PROGRAM MAIN
VAR
		// stepper function blocks  
	mcPower_1 : MC_Power;
	mcReset_1 : MC_Reset;
	mcJogging_1 : MC_Jog;
	mcMoveAbs_1 : MC_MoveAbsolute;
	mcMoveRel_1 : MC_MoveRelative;
	mcStop : MC_Stop;
	mcHome_1 : MC_Home;
	
	bEnableAxis_1 : BOOL;
	bJogForwards : BOOL;
	bJogBackwards: BOOL;
	eJogMode : E_JogMode; 
	bMoveDone : BOOL;	
	bAbsMove: BOOL;
	bRelMove: BOOL;
	
	heartbeat: BYTE; 
	//FbStageMotion : FB_Stage_Motion;

	bStop: BOOL;
	bHomeAxis_1: BOOL;

	// action Variables
	mcMoveAbsTest_1 : MC_MoveAbsolute;
	mcMoveAbsTestReturn_1 : MC_MoveAbsolute;
	iState : DINT;
	bStartTest : BOOL;
	bFinishTest: BOOL;
	fbReturnTimer : TON; // timer delay for the cycle to return home.
	fbDutyCycleTimer : TON; // timer duty cycle so the delay between cycles
	bStartReturnTimer : BOOL;
	bStartDutyCycleTimer : BOOL;	
	fbTestCycleCounter  : CTU;
	bCycleComplete : BOOL;
	bCycleCounterReset : BOOL;
	bTestFinished : BOOL;
	bTestRelMove: BOOL;
	
	bEnableAxisPosative_1: BOOL;
	bEnableAxisNegative_1: BOOL;
END_VAR

VAR_INPUT
	fAbsPos_1: LREAL;
	fRelDistance: LREAL;
	fRelTestDistance: LREAL;
	fAbsTestDistance: LREAL;
	fHomePosition: LREAL;
	fAxisVelocity: LREAL;
	fAxisAcceleration: LREAL;
	
// action Variables
	iCycleCount : WORD;
	fReturnTime : TIME;
	uInputReurnTime : UINT;
	fDutyCycleTime : TIME;
	uInputCycleTime : UINT;
	fTempLimit : DINT;
	
// Digital Inputs
	LimitSwitchInput_1 AT %I* : BOOL;
	LimitSwitchInput_2 AT %I* : BOOL;
	
// Analouge Inputs
	ThermoCoupleValue_Ch1 AT %I* : DINT;  
END_VAR

VAR_OUTPUT
// action Variables	
	iCurrentCycleValue : WORD;
		// Digital outputs
	LimitSwitchOutput_1 AT %Q* : BOOL;
	LimitSwitchOutput_2 AT %Q* : BOOL;
	EncoderPowerOutput_3 AT %Q* : BOOL;
	EncoderPowerOutput_6 AT %Q* : BOOL;
END_VAR

heartbeat := heartbeat + 1;

Limit_Switch();
Thermo_Couple();
EncoderPowerOutput_3 := TRUE;
EncoderPowerOutput_6 := TRUE;

mcStop(Axis := GVL.stAxis_1, Execute := bStop,);

mcPower_1(Axis := GVL.stAxis_1, Enable := bEnableAxis_1, Enable_Positive := bEnableAxisPosative_1, Enable_Negative := bEnableAxisNegative_1, Override := 100.0);

mcReset_1(Axis := GVL.stAxis_1, Execute := NOT(bEnableAxis_1));

mcJogging_1(Axis := GVL.stAxis_1, JogForward := bJogForwards, JogBackwards := bJogBackwards, Velocity := fAxisVelocity, Acceleration := fAxisAcceleration, Deceleration := fAxisAcceleration, Jerk := 0.8);

mcMoveAbs_1 (Axis := GVL.stAxis_1, Execute := bAbsMove, Position := fAbsPos_1, Velocity := fAxisVelocity, Acceleration := fAxisAcceleration, Deceleration := fAxisAcceleration);
bAbsMove := FALSE;

mcMoveRel_1(Axis := GVL.stAxis_1, Execute := bRelMove, Distance := fRelDistance, Velocity := fAxisVelocity, Acceleration := fAxisAcceleration, Deceleration := fAxisAcceleration);
bRelMove := FALSE;

//mcHome_1(Axis := GVL.stAxis_1, Execute := bHomeAxis_1, Position := fHomePosition);


Test_Routine();

ACTION Limit_Switch:
LimitSwitchOutput_1 := TRUE;
LimitSwitchOutput_2 := TRUE;

IF LimitSwitchInput_1 THEN
	bEnableAxisPosative_1 := TRUE;
ELSE
	bEnableAxisPosative_1 := FALSE ;	
	
END_IF

IF LimitSwitchInput_2 THEN
	bEnableAxisNegative_1 := TRUE;
ELSE
	bEnableAxisNegative_1 := FALSE ;	
	
END_IF
END_ACTION

ACTION Test_Routine:
mcMoveAbsTest_1(Axis := GVL.stAxis_1, Position := 10, Velocity := fAxisVelocity, Acceleration := fAxisAcceleration, Deceleration := fAxisAcceleration);	
mcMoveAbsTest_1.Execute := FALSE;
fbReturnTimer( IN := bStartReturnTimer, PT := fReturnTime);	
mcMoveAbsTestReturn_1(Axis := GVL.stAxis_1, Position := 0, Velocity := fAxisVelocity, Acceleration := fAxisAcceleration, Deceleration := fAxisAcceleration);
mcMoveAbsTestReturn_1.Execute := FALSE;
fbReturnTimer( IN := bStartReturnTimer, PT := fReturnTime);	
fbDutyCycleTimer( IN := bStartDutyCycleTimer, PT := fDutyCycleTime);	
fbTestCycleCounter(CU := bCycleComplete, RESET := bCycleCounterReset, PV := iCycleCount);
fReturnTime:= INT_TO_TIME(uInputReurnTime);
fDutyCycleTime:= INT_TO_TIME(uInputCycleTime);
CASE iState OF
	
	// initialising the state machine so starting a homing rotuine reseting the counter to 0 
	0: 
		iState := 10;
	10: 
		IF bStartTest THEN
			iState := 20;
		END_IF
	
	20:
	
		mcMoveAbsTest_1.Execute := TRUE;
		IF mcMoveAbsTest_1.Done THEN
			bStartReturnTimer := TRUE;
			iState := 30;
		END_IF

	30:
		fbReturnTimer( IN := bStartReturnTimer, PT := fReturnTime);	
		IF MAIN.fbReturnTimer.Q THEN
			bStartReturnTimer := FALSE;
			iState := 40;
		END_IF
	

	40:
		mcMoveAbsTestReturn_1.Execute := TRUE;
		IF mcMoveAbsTestReturn_1.Done THEN
			bStartDutyCycleTimer := TRUE;
			iState := 50;
		END_IF	
	
	50:
		fbDutyCycleTimer( IN := bStartDutyCycleTimer, PT := fDutyCycleTime);	
		IF MAIN.fbDutyCycleTimer.Q THEN
			bStartDutyCycleTimer := FALSE;
			iState := 60;
		END_IF

	60: bCycleComplete := TRUE;
		iState := 70;
	
	70: fbTestCycleCounter(CU := bCycleComplete, RESET := bCycleCounterReset, PV := iCycleCount);
		IF MAIN.fbTestCycleCounter.Q THEN
			iState := 90; 
		ELSE
		bCycleComplete := FALSE;	
		iState := 20;
		END_IF
	
	90: bStartTest := FALSE;
		bFinishTest := TRUE;
		iState := 10;
	
ELSE
	;
END_CASE
END_ACTION

ACTION Thermo_Couple:
	IF ThermoCoupleValue_Ch1 >= fTempLimit THEN
		mcstop.Execute := TRUE; 
	ELSE
		mcstop.Execute := FALSE; 
	END_IF
END_ACTION

END_PROGRAM

(* stored: Version 1.1.0.1, ProductVersion 3.1.4024.0
   POU MAIN: Id {ed9b3e07-4467-47c3-9766-2d2ed915d21b}, SpecialFunc None
   Action Limit_Switch: Id {b3b7bac8-26ca-4866-bea2-1a68ac32b6f9}
   Action Test_Routine: Id {63bc1eb6-c2bb-4839-87a7-c55c6bea2977}
   Action Thermo_Couple: Id {6678029e-6d8f-4c39-9a51-29de60c369fe} *)
